{attribute 'GeneratedUsingTerminal: EL3773-0000-0018'}
{attribute addProperty BoxType "EL3773-0000-0018"}
{attribute addProperty Id "U3_StatusAT %I*U3_Status_DC9039207"}
{attribute addProperty CRC "658469525"}
{attribute addProperty Size "7"}
TYPE L3_Voltage_Status_273F7295 EXTENDS InputBase_8311D824 :
STRUCT
	{attribute addProperty Name "U3_Status"}
	U3_Status AT %I* : U3_Status_DC903920;
END_STRUCT
END_TYPE

(* stored: Version 1.2.0.0, ProductVersion 3.1.4024.9
   DUT L3_Voltage_Status_273F7295: Id {e9cf81ae-871f-4db7-96c7-42ad4b4ee528} *)
